// TIA Portal V19 export
TYPE "LAF_typeChecksumCatBool"
TITLE = Structure PLC checksum cat bool / Struktur PLC checksum cat Bool
// Type contains the structure for edge evaluations / PLC checksum
// stored: Access Published
   STRUCT
      standard { ExternalAccessible := 'False'; ExternalVisible := 'False'; ExternalWritable := 'False'} : Bool;   // Standard
      safety { ExternalAccessible := 'False'; ExternalVisible := 'False'; ExternalWritable := 'False'} : Bool;   // Safety
      textlists { ExternalAccessible := 'False'; ExternalVisible := 'False'; ExternalWritable := 'False'} : Bool;   // Textlisten / Textlists
   END_STRUCT;
END_TYPE
